SUBAPPLICATION Dom (* Subapplication Type *)
  (* Standard: 61499-2 *)
  (* Version 1.0, 2023-01-29, Franz *)
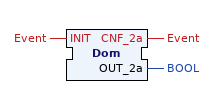
  EVENT_INPUT
    INIT;
  END_EVENT
  EVENT_OUTPUT
    CNF_2a;
  END_EVENT
  VAR_OUTPUT
    OUT_2a : BOOL;
  END_VAR
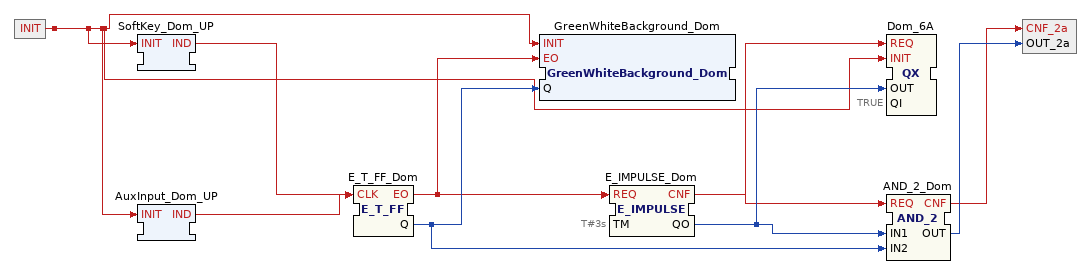
  FBS
    AND_2_Dom : AND_2;
    E_T_FF_Dom : E_T_FF;
    Dom_6A : QX(QI := TRUE);
    E_IMPULSE_Dom : E_IMPULSE(TM := T#3s);
  END_FBS
  SUBAPPS
    GreenWhiteBackground_Dom : GreenWhiteBackground_Dom;
  END_SUBAPPS
  SUBAPPLICATION AuxInput_Dom_UP
    EVENT_INPUT
      INIT;
    END_EVENT
    EVENT_OUTPUT
      IND;
    END_EVENT
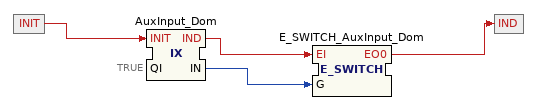
    FBS
      E_SWITCH_AuxInput_Dom : E_SWITCH;
      AuxInput_Dom : IX(QI := TRUE);
    END_FBS
    EVENT_CONNECTIONS
      AuxInput_Dom.IND TO E_SWITCH_AuxInput_Dom.EI;
      INIT TO AuxInput_Dom.INIT;
      E_SWITCH_AuxInput_Dom.EO0 TO IND;
    END_CONNECTIONS
    DATA_CONNECTIONS
      AuxInput_Dom.IN TO E_SWITCH_AuxInput_Dom.G;
    END_CONNECTIONS
  END_SUBAPPLICATION
  SUBAPPLICATION SoftKey_Dom_UP
    EVENT_INPUT
      INIT;
    END_EVENT
    EVENT_OUTPUT
      IND;
    END_EVENT
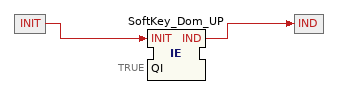
    FBS
      SoftKey_Dom_UP : IE(QI := TRUE);
    END_FBS
    EVENT_CONNECTIONS
      INIT TO SoftKey_Dom_UP.INIT;
      SoftKey_Dom_UP.IND TO IND;
    END_CONNECTIONS
  END_SUBAPPLICATION
  EVENT_CONNECTIONS
    E_IMPULSE_Dom.CNF TO AND_2_Dom.REQ;
    E_T_FF_Dom.EO TO E_IMPULSE_Dom.REQ;
    E_IMPULSE_Dom.CNF TO Dom_6A.REQ;
    AND_2_Dom.CNF TO CNF_2a;
    INIT TO SoftKey_Dom_UP.INIT;
    SoftKey_Dom_UP.IND TO E_T_FF_Dom.CLK;
    INIT TO AuxInput_Dom_UP.INIT;
    AuxInput_Dom_UP.IND TO E_T_FF_Dom.CLK;
    INIT TO Dom_6A.INIT;
    INIT TO GreenWhiteBackground_Dom.INIT;
    E_T_FF_Dom.EO TO GreenWhiteBackground_Dom.EO;
  END_CONNECTIONS
  DATA_CONNECTIONS
    E_IMPULSE_Dom.QO TO AND_2_Dom.IN1;
    E_T_FF_Dom.Q TO AND_2_Dom.IN2;
    E_IMPULSE_Dom.QO TO Dom_6A.OUT;
    AND_2_Dom.OUT TO OUT_2a;
    E_T_FF_Dom.Q TO GreenWhiteBackground_Dom.Q;
  END_CONNECTIONS
END_SUBAPPLICATION
